FUNCTION Matrix_SameSizeAs_Array2D : BOOL
VAR_IN_OUT
	A : ARRAY[*,*] OF LREAL;
END_VAR
VAR_INPUT
	M : REFERENCE TO Matrix;
END_VAR

//check for bad references
IF NOT(__ISVALIDREF(M)) THEN
	Matrix_SameSizeAs_Array2D := FALSE;
	RETURN;
END_IF

//check for size mismatch
Matrix_SameSizeAs_Array2D := Array2D_Rows(A) = M.Rows AND Array2D_Cols(A) = M.Cols;

END_FUNCTION

(* stored: Version 1.1.0.1, ProductVersion 3.1.4024.9
   POU Matrix_SameSizeAs_Array2D: Id {c9358c1e-1fa6-0af9-1809-136157085d7a}, SpecialFunc None *)
